FUNCTION_BLOCK Randn (* Function Block For Level Sensor *)
  (* Standard: 61499-2 *)
  (* Version 0.0, 2018-01-22, Duc Do Tran, OFFIS e.V. *)
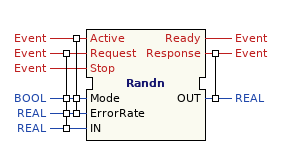
  EVENT_INPUT
    Active WITH ErrorRate, Mode; (* Initialization Request *)
    Request WITH IN, ErrorRate, Mode; (* Normal Execution Request *)
    Stop;
  END_EVENT
  EVENT_OUTPUT
    Ready; (* Initialization Confirm *)
    Response WITH OUT; (* Execution Confirmation *)
  END_EVENT
  VAR_INPUT
    Mode : BOOL; (* 0 : Error in (% ); 1 : Error in (+-) *)
    ErrorRate : REAL := 0.05; (* Error rate of Sensor *)
    IN : REAL; (* set value *)
  END_VAR
  VAR_OUTPUT
    OUT : REAL; (* Signal for controller *)
  END_VAR
  VAR
    RandNum : UINT; (* Internal Variable *)
    ErrorR : REAL; (* Internal Variable *)
  END_VAR
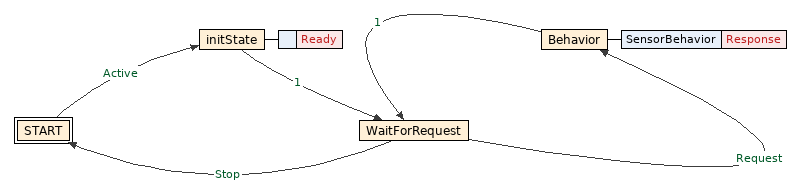
  EC_STATES
    START; (* Initial State *)
    Behavior : SensorBehavior -> Response;
    initState : -> Ready;
    WaitForRequest;
  END_STATES
  EC_TRANSITIONS
    START TO initState := Active;
    Behavior TO WaitForRequest := 1;
    WaitForRequest TO Behavior := Request;
    WaitForRequest TO START := Stop;
    initState TO WaitForRequest := 1;
  END_TRANSITIONS
  ALGORITHM SensorBehavior IN ST: (* new algorithm *)
RandNum := rand()  MOD 1000;
ErrorR := ErrorRate * (2 * UINT_TO_REAL(RandNum)/1000 - 1);
IF (Mode = TRUE) THEN
	OUT := IN + ErrorR;
ELSE
	OUT := IN*(1 - ErrorR);
END_IF;
  END_ALGORITHM
END_FUNCTION_BLOCK
